TYPE ST_AxisInterlock :
STRUCT
END_STRUCT
END_TYPE

(* stored: Version 1.1.0.1, ProductVersion 3.1.4026.18
   DUT ST_AxisInterlock: Id {b89579d9-5006-4b18-b612-28926a53fc50} *)
